SYSTEM ClientTest
  APPLICATION ClientTestApp
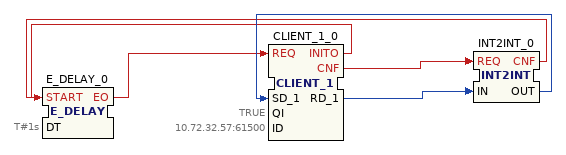
    FBS
      CLIENT_1_0 : CLIENT_1(QI := TRUE, ID := 10.72.32.57:61500);
      INT2INT_0 : INT2INT;
      E_DELAY_0 : E_DELAY(DT := T#1s);
    END_FBS
    EVENT_CONNECTIONS
      E_DELAY_0.EO TO CLIENT_1_0.REQ;
      CLIENT_1_0.INITO TO E_DELAY_0.START;
      CLIENT_1_0.CNF TO INT2INT_0.REQ;
      INT2INT_0.CNF TO E_DELAY_0.START;
    END_CONNECTIONS
    DATA_CONNECTIONS
      CLIENT_1_0.RD_1 TO INT2INT_0.IN;
      INT2INT_0.OUT TO CLIENT_1_0.SD_1;
    END_CONNECTIONS
  END_APPLICATION
  DEVICE FORTE_PC_1 : FORTE_PC(MGR_ID := "localhost:61499")
    {SET_ATTRIBUTE(Profile, HOLOBLOC)}
    RESOURCE EMB_RES : EMB_RES
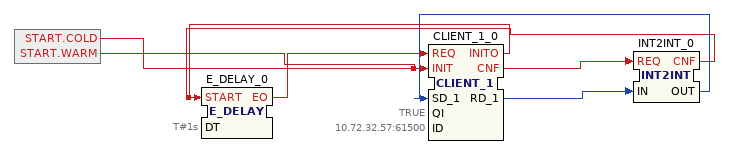
      FBS
        E_DELAY_0 : E_DELAY(DT := T#1s);
        CLIENT_1_0 : CLIENT_1(QI := TRUE, ID := 10.72.32.57:61500);
        INT2INT_0 : INT2INT;
      END_FBS
      EVENT_CONNECTIONS
        E_DELAY_0.EO TO CLIENT_1_0.REQ;
        CLIENT_1_0.INITO TO E_DELAY_0.START;
        CLIENT_1_0.CNF TO INT2INT_0.REQ;
        INT2INT_0.CNF TO E_DELAY_0.START;
        START.COLD TO CLIENT_1_0.INIT;
        START.WARM TO CLIENT_1_0.INIT;
      END_CONNECTIONS
      DATA_CONNECTIONS
        CLIENT_1_0.RD_1 TO INT2INT_0.IN;
        INT2INT_0.OUT TO CLIENT_1_0.SD_1;
      END_CONNECTIONS
    END_RESOURCE
  END_DEVICE
  MAPPINGS
    ClientTestApp.CLIENT_1_0 ON FORTE_PC_1.EMB_RES.CLIENT_1_0;
    ClientTestApp.INT2INT_0 ON FORTE_PC_1.EMB_RES.INT2INT_0;
    ClientTestApp.E_DELAY_0 ON FORTE_PC_1.EMB_RES.E_DELAY_0;
  END_MAPPINGS
  SEGMENTS
    Ethernet : Ethernet;
  END_SEGMENTS
  LINKS
    FORTE_PC_1 => Ethernet;
  END_LINKS
END_SYSTEM
